{attribute addProperty BoxType "EP1312-0001-0016"}
{attribute addProperty Id "A_0038_EP1518_0002_0016EP1518_1EB154A835444.25A_0039_EP1518_0002_0017EP1518_1EB154A835444.25A_0040_EP1518_0002_0018EP1518_1EB154A835444.25A_0041_EP1518_0002_0019EP1518_1EB154A835444.25A_0042_EP1809_0021_0016EP1809_248EAA3414618.25A_0043_EP1809_0021_0017EP1809_248EAA3414618.25A_0044_EP1809_0022_0017EP1809_248EAA3414618.25A_0045_EP1809_0022_0018EP1809_248EAA3414618.25A_0046_EP1809_0042_0018EP1809_4E090DF614618.25A_0047_EP1809_0042_0019EP1809_09F99349429496725034359738362.25A_0048_EP1816_0003_0016EP1816_8758F16324230.25A_0049_EP1816_0008_0016EP1816_5EE46DF622628.25A_0050_EP1816_0008_0017EP1816_5EE46DF622628.25A_0051_EP1816_0008_0018EP1816_C79E751722628.25A_0052_EP1816_0008_0019EP1816_C79E751722628.25A_0053_EP1816_0008_0020EP1816_C79E751722628.25A_0054_EP1816_1008_0016EP1816_CEA0212F24230.25A_0055_EP1816_1008_0017EP1816_CEA0212F24230.25A_0056_EP1816_3008_0016EP1816_F6DE3BA643454.25A_0057_EP1816_3008_0017EP1816_F6DE3BA643454.25A_0058_EP1816_3008_0018EP1816_F6DE3BA643454.25A_0059_EP1819_0021_0016EP1819_248EAA3414618.25A_0060_EP1819_0021_0017EP1819_248EAA3414618.25A_0061_EP1819_0022_0016EP1819_248EAA3414618.25A_0062_EP1819_0022_0017EP1819_248EAA3414618.25A_0063_EP1859_0042_0018EP1859_AFA720D514618.25A_0064_EP1859_0042_0019EP1859_B48C22F8429496725034359738362.25"}
{attribute addProperty CRC "2447648170"}
{attribute addProperty SizeInBites "5942"}
{attribute addProperty SizeInBytes "68719477478.75"}
TYPE A_0037_EP1312_0001_0016_91E425AA EXTENDS EP1312_179A0949 :
STRUCT
	{attribute addProperty Name "A_0038_EP1518_0002_0016"}
	A_0038_EP1518_0002_0016 : EP1518_1EB154A8;
	{attribute addProperty Name "A_0039_EP1518_0002_0017"}
	A_0039_EP1518_0002_0017 : EP1518_1EB154A8;
	{attribute addProperty Name "A_0040_EP1518_0002_0018"}
	A_0040_EP1518_0002_0018 : EP1518_1EB154A8;
	{attribute addProperty Name "A_0041_EP1518_0002_0019"}
	A_0041_EP1518_0002_0019 : EP1518_1EB154A8;
	{attribute addProperty Name "A_0042_EP1809_0021_0016"}
	A_0042_EP1809_0021_0016 : EP1809_248EAA34;
	{attribute addProperty Name "A_0043_EP1809_0021_0017"}
	A_0043_EP1809_0021_0017 : EP1809_248EAA34;
	{attribute addProperty Name "A_0044_EP1809_0022_0017"}
	A_0044_EP1809_0022_0017 : EP1809_248EAA34;
	{attribute addProperty Name "A_0045_EP1809_0022_0018"}
	A_0045_EP1809_0022_0018 : EP1809_248EAA34;
	{attribute addProperty Name "A_0046_EP1809_0042_0018"}
	A_0046_EP1809_0042_0018 : EP1809_4E090DF6;
	{attribute addProperty Name "A_0047_EP1809_0042_0019"}
	A_0047_EP1809_0042_0019 : EP1809_09F99349;
	{attribute addProperty Name "A_0048_EP1816_0003_0016"}
	A_0048_EP1816_0003_0016 : EP1816_8758F163;
	{attribute addProperty Name "A_0049_EP1816_0008_0016"}
	A_0049_EP1816_0008_0016 : EP1816_5EE46DF6;
	{attribute addProperty Name "A_0050_EP1816_0008_0017"}
	A_0050_EP1816_0008_0017 : EP1816_5EE46DF6;
	{attribute addProperty Name "A_0051_EP1816_0008_0018"}
	A_0051_EP1816_0008_0018 : EP1816_C79E7517;
	{attribute addProperty Name "A_0052_EP1816_0008_0019"}
	A_0052_EP1816_0008_0019 : EP1816_C79E7517;
	{attribute addProperty Name "A_0053_EP1816_0008_0020"}
	A_0053_EP1816_0008_0020 : EP1816_C79E7517;
	{attribute addProperty Name "A_0054_EP1816_1008_0016"}
	A_0054_EP1816_1008_0016 : EP1816_CEA0212F;
	{attribute addProperty Name "A_0055_EP1816_1008_0017"}
	A_0055_EP1816_1008_0017 : EP1816_CEA0212F;
	{attribute addProperty Name "A_0056_EP1816_3008_0016"}
	A_0056_EP1816_3008_0016 : EP1816_F6DE3BA6;
	{attribute addProperty Name "A_0057_EP1816_3008_0017"}
	A_0057_EP1816_3008_0017 : EP1816_F6DE3BA6;
	{attribute addProperty Name "A_0058_EP1816_3008_0018"}
	A_0058_EP1816_3008_0018 : EP1816_F6DE3BA6;
	{attribute addProperty Name "A_0059_EP1819_0021_0016"}
	A_0059_EP1819_0021_0016 : EP1819_248EAA34;
	{attribute addProperty Name "A_0060_EP1819_0021_0017"}
	A_0060_EP1819_0021_0017 : EP1819_248EAA34;
	{attribute addProperty Name "A_0061_EP1819_0022_0016"}
	A_0061_EP1819_0022_0016 : EP1819_248EAA34;
	{attribute addProperty Name "A_0062_EP1819_0022_0017"}
	A_0062_EP1819_0022_0017 : EP1819_248EAA34;
	{attribute addProperty Name "A_0063_EP1859_0042_0018"}
	A_0063_EP1859_0042_0018 : EP1859_AFA720D5;
	{attribute addProperty Name "A_0064_EP1859_0042_0019"}
	A_0064_EP1859_0042_0019 : EP1859_B48C22F8;
END_STRUCT
END_TYPE

(* stored: Version 1.2.0.0, ProductVersion 3.1.4024.9
   DUT A_0037_EP1312_0001_0016_91E425AA: Id {d21cd98e-fe4e-4236-a0a9-b5e721b68625} *)
